(* IEC 61131-3 sources: POMIRTS_lab3/AS/Library_2/DRVABDF1, 3 files *)

(* ---- DRVABDF1.typ ---- *)
TYPE

END_TYPE

(* ---- DRVABDF1.fun ---- *)
{REDUND_CONTEXT} {REDUND_UNREPLICABLE}  FUNCTION_BLOCK ABDF1Master			(*operates the DF1 protocol (full-duplex) at runtime*)
	VAR_INPUT
		enable	:BOOL;				(*enables execution*)
		ident	:UDINT;				(*ident from the ABDF1MOpen() FBK*)
	END_VAR
	VAR_OUTPUT
		status	:UINT;				(*execution status: ERR_OK, ERR_FUB_ENABLE_FALSE, 0xXXXX = see help*)
		execute	:BOOL;				(*command was executed (execute = 1)*)
		recordnum	:UINT;			(*number of the entry in the data object currently being processed*)
		sts	:USINT;					(*status byte (STS)*)
		ext_sts	:USINT;				(*extended status byte (EXT STS)*)
	END_VAR
END_FUNCTION_BLOCK

{REDUND_CONTEXT} {REDUND_UNREPLICABLE}  FUNCTION_BLOCK ABDF1MOpen
	VAR_INPUT
		enable	:BOOL;				(*enables execution*)
		pDevice	:UDINT;				(*device description string*)
		pMode	:UDINT;				(*mode description string*)
		pConfig	:UDINT;				(*data object name*)
		own_ID	:USINT;				(*own station number (0-254)*)
		checksum	:USINT;			(*checksum (BCC or CRC)*)
		timeout	:UINT;				(*timeout in milliseconds (multiple of 10)*)
	END_VAR
	VAR_OUTPUT
		status	:UINT;				(*execution status: ERR_OK, ERR_FUB_ENABLE_FALSE, 0xXXXX = see help*)
		ident	:UDINT;				(*ident*)
	END_VAR
END_FUNCTION_BLOCK

{REDUND_CONTEXT} {REDUND_UNREPLICABLE}  FUNCTION_BLOCK ABDF1SOpen			(*returns the ident for ABDF1Slave(), ABDF1SClose(), ABDF1Master() and ABDF1MClose()*)
	VAR_INPUT
		enable	:BOOL;				(*enables execution*)
		pDevice	:UDINT;				(*device description string*)
		pMode	:UDINT;				(*mode description string*)
		pConfig	:UDINT;				(*name of a data object*)
		own_ID	:USINT;				(*own node number (0-254)*)
		checksum	:USINT;			(*checksum (BCC or CRC)*)
		timeout	:UINT;				(*timeout in milliseconds (multiple of 10)*)
	END_VAR
	VAR_OUTPUT
		status	:UINT;				(*execution status: ERR_OK, ERR_FUB_ENABLE_FALSE, 0xXXXX = see help*)
		ident	:UDINT;				(*ident*)
	END_VAR
END_FUNCTION_BLOCK

{REDUND_CONTEXT} {REDUND_UNREPLICABLE}  FUNCTION_BLOCK ABDF1Slave			(*operates the DF1 protocol (full-duplex) at runtime*)
	VAR_INPUT
		enable	:BOOL;				(*enables execution*)
		ident	:UDINT;				(*ident from the ABDF1SOpen() FBK*)
	END_VAR
	VAR_OUTPUT
		status	:UINT;				(*execution status: ERR_OK, ERR_FUB_ENABLE_FALSE, 0xXXXX = see help*)
		exec	:UINT;				(*counter for DF1 commands received*)
		cmd	:USINT;					(*last received command*)
		fct	:USINT;					(*last received function*)
		len	:UDINT;					(*length of the data to be copied*)
	END_VAR
END_FUNCTION_BLOCK

{REDUND_CONTEXT} {REDUND_UNREPLICABLE}  FUNCTION_BLOCK ABDF1SClose			(*closes the driver environment, after which the ABDF1SOpen() FBK can be called again*)
	VAR_INPUT
		enable	:BOOL;				(*enables execution*)
		ident	:UDINT;				(*ident from the ABDF1SOpen() FBK*)
	END_VAR
	VAR_OUTPUT
		status	:UINT;				(*execution status: ERR_OK, ERR_FUB_ENABLE_FALSE, 0xXXXX = see help*)
	END_VAR
END_FUNCTION_BLOCK

{REDUND_CONTEXT} {REDUND_UNREPLICABLE}  FUNCTION_BLOCK ABDF1MClose			(*closes the driver environment, after which the ABDF1MOpen() FBK can be called again*)
	VAR_INPUT
		enable	:BOOL;				(*enables execution*)
		ident	:UDINT;				(*ident from the ABDF1MOpen() FBK*)
	END_VAR
	VAR_OUTPUT
		status	:UINT;				(*execution status: ERR_OK, ERR_FUB_ENABLE_FALSE, 0xXXXX = see help*)
	END_VAR
END_FUNCTION_BLOCK

(* ---- DRVABDF1.var ---- *)
VAR CONSTANT
	df1ERR_CFG_LOCALPV	: UINT	:= 30064;			(*invalid LocalPV specified in data object*)
	df1ERR_CFG_EVENTPV	: UINT	:= 30061;			(*invalid EventPV specified in data object*)
	df1ERR_ILG_OWN_ID	: UINT	:= 30051;			(*invalid station number*)
	df1ERR_ILG_DEVICE	: UINT	:= 30055;			(*device already being used as a master/slave or invalid device string*)
	df1ERR_CFG_REMOTE	: UINT	:= 30065;			(*invalid remote addressing in data object*)
	df1ERR_CFG_LENGTH	: UINT	:= 30066;			(*invalid length specified in data object*)
	df1ERR_ILG_IDENT	: UINT	:= 30054;			(*invalid ident*)
	df1ERR_ILG_FRAME	: UINT	:= 30080;			(*invalid frame (no DF1 protocol)*)
	df1ERR_FRM_WRITE	: UINT	:= 30073;			(*error writing a frame (FRM_write())*)
	df1ERR_FRM_CLOSE	: UINT	:= 30074;			(*error closing the interface (FRM_close())*)
	df1ERR_CFG_ENTRY	: UINT	:= 30060;			(*incorrect entry or format in data object*)
	df1ERR_FRM_READ	: UINT	:= 30070;				(*error receiving frame (FRM_read())*)
	df1ERR_FRM_RBUF	: UINT	:= 30071;				(*error in buffer return (FRM_rbuf())*)
	df1ERR_FRM_GBUF	: UINT	:= 30072;				(*no write buffer available (FRM_gbuf())*)
	df1ERR_CHECKSUM	: UINT	:= 30053;				(*invalid or unsupported checksums*)
	df1CHECKSUM_CRC	: USINT	:= 0;					(*CRC checksum calculation (Cyclic Redundancy Check)*)
	df1CHECKSUM_BCC	: USINT	:= 1;					(*BCC checksum calculation*)
	df1ERR_TIMEOUT	: UINT	:= 30052;				(*invalid timeout time or timeout time exceeded*)
	df1ERR_ILG_CFG	: UINT	:= 30050;				(*data object doesn't exist*)
	df1ERR_COMMAND	: UINT	:= 30081;				(*invalid request (COMMAND)*)
	df1ERR_CFG_STN	: UINT	:= 30063;				(*invalid station number specified; broadcasts not supported*)
	df1ERR_CFG_CMD	: UINT	:= 30062;				(*invalid command or function code specified; command not supported*)
	df1ERR_MEMORY	: UINT	:= 30085;				(*no memory available for driver management or error freeing memory*)
	df1ERR_REPLY	: UINT	:= 30082;				(*invalid response (REPLY)*)
	df1ERR_NAK	: UINT	:= 30083;					(*max. number of NAKs (negative acknowledgements) reached*)
	df1ERR_ENQ	: UINT	:= 30084;					(*max. number of ENQs (queries) reached*)
END_VAR
